// TIA Portal V17 export
// export: Created 2022-06-18T17:45:09.1477249Z, ExportSetting None, DisplayName Totally Integrated Automation Portal, DisplayVersion V17, DisplayName TIA Portal Openness, DisplayVersion V17, DisplayName TIA Portal Teamcenter Gateway, DisplayVersion V17, DisplayName TIA Portal Version Control Interface, DisplayVersion V17, DisplayName TIA Portal Test Suite Advanced, DisplayVersion V17, DisplayName SINAMICS Startdrive Advanced, DisplayVersion V17, DisplayName SINAMICS DCC, DisplayVersion V17, DisplayName SINAMICS Startdrive G130, G150, S120, S150, SINAMICS MV, S210, DisplayVersion V17, DisplayName SINAMICS Startdrive G110M, G120, G120C, G120D, G120P, G115D, DisplayVersion V17, DisplayName STEP 7 Professional, DisplayVersion V17, DisplayName SIMATIC Energy Suite, DisplayVersion V17, DisplayName STEP 7 CFC, DisplayVersion V17, DisplayName STEP 7 Safety, DisplayVersion V17, DisplayName WinCC Advanced / Unified PC, DisplayVersion V17, DisplayName SIMATIC Visualization Architect, DisplayVersion V17
DATA_BLOCK "GlobalDB"   // DB999
TITLE = TetsTitle
{ S7_Optimized_Access := 'TRUE' }
AUTHOR : AV
FAMILY : TestFamily
NAME : Q741P
VERSION : 0.11
// Test Comment
// stored: MemoryReserve 100
   VAR
      i_VarInt : Int;
      r_VarReal : Real;
      VarBool : Bool;
      VarBoolTest : Bool;
      VarUDT : "Lib_UDT_Motor_DS_RotSens";
   END_VAR
BEGIN
END_DATA_BLOCK
